// TIA Portal project "Pick & Place XYZ" (V15.1)
// Vorlageprojekt für das Buch mit Zielsystem S7-1200

(* hardware
DEVICE "S7-1200-Station_1"  S7-1200 Station
   slot 0: "Baugruppenträger_0"  Rack  V1.0
   slot 1: "PLC_1"  CPU 1214C DC/DC/DC  6ES7 214-1AG40-0XB0  V4.2
*)

// ===== PLC "PLC_1"  CPU 1214C DC/DC/DC =====

VAR_GLOBAL   // PLC tag table "Standard-Variablentabelle"
   "Transporte_caja" AT %Q0.1 : Bool;
   "Arranque" AT %I0.4 : Bool;
   "Caja_posicion" AT %I0.1 : Bool;
   "X" AT %ID30 : Real;
   "Y" AT %ID34 : Real;
   "Z" AT %ID38 : Real;
   "SPX" AT %QD30 : Real;
   "SPY" AT %QD34 : Real;
   "SPZ" AT %QD38 : Real;
   "Contador_caja" AT %QD42 : DInt;
   "Pallet_posicion" AT %I0.0 : Bool;
   "Sensor_robot" AT %I0.2 : Bool;
   "Sensor_limite-C" AT %I0.3 : Bool;
   "Reset" AT %I0.5 : Bool;
   "Paro" AT %I0.6 : Bool;
   "Paro emergencia" AT %I0.7 : Bool;
   "Automatico" AT %I1.0 : Bool;
   "Factori I/O" AT %I1.1 : Bool;
   "Transpote_pallet" AT %Q0.0 : Bool;
   "Transporte_salida" AT %Q0.2 : Bool;
   "Eje de rotacion" AT %Q0.3 : Bool;
   "Ventosa" AT %Q0.4 : Bool;
   "Baliza verde" AT %Q0.5 : Bool;
   "Baliza amarrila" AT %Q0.6 : Bool;
   "Baliza roja" AT %Q0.7 : Bool;
   "Luz_arranque" AT %Q1.0 : Bool;
   "Luz_reset" AT %Q1.1 : Bool;
   "Luz-paro" AT %Q1.2 : Bool;
   "ET0" AT %M100.0 : Bool;
   "Tag_1" AT %M250.0 : Bool;
   "ET1" AT %M100.1 : Bool;
   "BANDA LIBRE ET" AT %M300.0 : Bool;
   "ET2" AT %M100.2 : Bool;
   "Tag_2" AT %M250.1 : Bool;
   "ET3" AT %M100.3 : Bool;
   "PALLET CPL" AT %M300.1 : Bool;
   "ET4" AT %M100.4 : Bool;
   "ET5" AT %M100.5 : Bool;
   "ET6" AT %M100.6 : Bool;
   "TEMP1" AT %M300.2 : Bool;
   "ET7" AT %M100.7 : Bool;
   "ET8" AT %M101.0 : Bool;
   "ETI" AT %M99.7 : Bool;
   "TIPO CAJA" AT %MW50 : Int;
   "ET9" AT %M101.1 : Bool;
   "ET10" AT %M101.2 : Bool;
   "ET11" AT %M101.3 : Bool;
   "ET12" AT %M101.4 : Bool;
   "ET13" AT %M101.5 : Bool;
   "ET14" AT %M101.6 : Bool;
   "ET15" AT %M101.7 : Bool;
   "ET16" AT %M102.0 : Bool;
   "ET17" AT %M102.1 : Bool;
   "ET20" AT %M102.2 : Bool;
   "ET21" AT %M102.3 : Bool;
   "Tag_3" AT %M250.2 : Bool;
   "TEMP2" AT %M300.3 : Bool;
   "Tag_4" AT %M40.0 : Bool;
   "Marca_Arranque" AT %M60.0 : Bool;
   "Marca_paro" AT %M60.1 : Bool;
   "Marca_emergencia" AT %M60.2 : Bool;
END_VAR

// folder: System blocks/Program resources

DATA_BLOCK "IEC_Timer_0_DB"   // DB1
{ S7_Optimized_Access := 'TRUE' }
AUTHOR : Simatic
FAMILY : IEC
NAME : IEC_TMR
VERSION : 1.0
// stored: InstanceOfName IEC_TIMER
"IEC_TIMER"
BEGIN
END_DATA_BLOCK

DATA_BLOCK "IEC_Counter_0_DB"   // DB2
{ S7_Optimized_Access := 'TRUE' }
AUTHOR : Simatic
FAMILY : IEC
NAME : CNTR
VERSION : 1.0
// stored: InstanceOfName IEC_COUNTER
"IEC_COUNTER"
BEGIN
END_DATA_BLOCK

DATA_BLOCK "IEC_Timer_0_DB_1"   // DB3
{ S7_Optimized_Access := 'TRUE' }
AUTHOR : Simatic
FAMILY : IEC
NAME : IEC_TMR
VERSION : 1.0
// stored: InstanceOfName IEC_TIMER
"IEC_TIMER"
BEGIN
END_DATA_BLOCK

DATA_BLOCK "IEC_Counter_0_DB_1"   // DB4
{ S7_Optimized_Access := 'TRUE' }
AUTHOR : Simatic
FAMILY : IEC
NAME : CNTR
VERSION : 1.0
// stored: InstanceOfName IEC_COUNTER
"IEC_COUNTER"
BEGIN
END_DATA_BLOCK

// folder: (top level)

FUNCTION "MHJ-PLC-Lab-Function-S71200" : Void   // FC9000, SCL
{ S7_Optimized_Access := 'TRUE' }
VERSION : 0.1
   VAR_TEMP
      rdTimeReturn : Int;
      outputTime : DTL;
      SyncVal : Byte;
      forVal : Int;
      forVal_2 : Int;
      Value : Byte;
   END_VAR
   VAR CONSTANT
      CompVal : Byte := 16#34;
      Value_01 : Byte := 16#11;
      Value_01_DW : DWord := 16#A165_D992;
      Value_02_DW : DWord := 16#58BE_4401;
   END_VAR
BEGIN

   #Value:=PEEK(area := 16#82,
        dbNumber := 0,
        byteOffset := 511);
   #Value := #Value + 1;

   POKE(area := 16#82,
        dbNumber := 0,
        byteOffset := 511,
        value := #Value);

   POKE(area:=16#81,
        dbNumber:=0,
        byteOffset:=1016,
        value:=#Value_01_DW);
   POKE(area := 16#81,
        dbNumber := 0,
        byteOffset := 1020,
        value := #Value_02_DW);

   POKE(area := 16#81,
        dbNumber := 0,
        byteOffset := 511,
        value := B#16#00);

   FOR #forVal := 0 TO 120 DO
       FOR #forVal_2:=0 TO 10 DO
           #rdTimeReturn:=RD_SYS_T(#outputTime);
           #rdTimeReturn := WR_SYS_T(#outputTime);
           #rdTimeReturn := RD_SYS_T(#outputTime);
           #rdTimeReturn := WR_SYS_T(#outputTime);
       END_FOR;
       #SyncVal:= PEEK(area := 16#81,
                      dbNumber := 0,
                      byteOffset := 511);
       IF #SyncVal = #CompVal THEN
          GOTO M_1;
       END_IF;
   END_FOR;
   RETURN;

   M_1:
   POKE(area := 16#81,
        dbNumber := 0,
        byteOffset := 511,
        value := B#16#0);
END_FUNCTION

ORGANIZATION_BLOCK "Main"   // OB1, LAD, ProgramCycle
TITLE = "Main Program Sweep (Cycle)"
{ S7_Optimized_Access := 'TRUE' }
VERSION : 0.1
   VAR_INPUT
      Initial_Call : Bool;   // Initial call of this OB
      Remanence : Bool;   // =True, if remanent data are available
   END_VAR
   VAR_TEMP   // added for the SCL form of the ladder/FBD networks
      _w1 : Bool;
      _w2 : Bool;
   END_VAR
BEGIN

REGION Network 1: Konnektierungsbaustein für PLC-Lab
   // Im Netzwerk 1 wird der Konnektierungsbaustein für PLC-Lab aufgerufen.
   // Dieser Aufruf darf nicht entfernt werden!
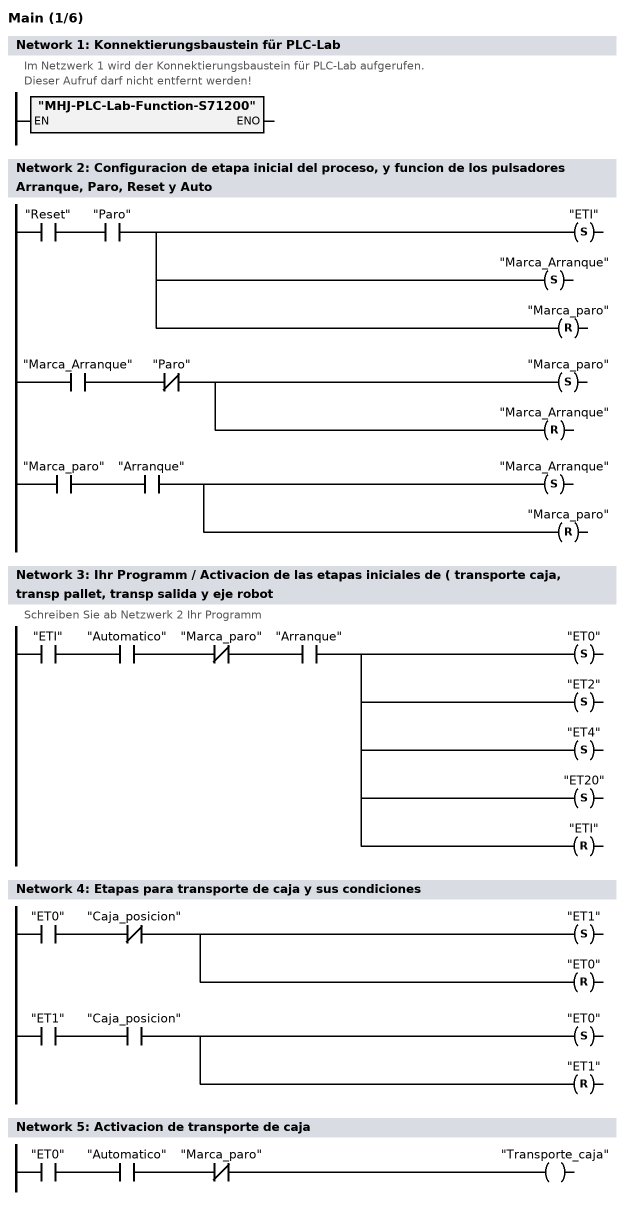
   RUNG wire#powerrail
      "MHJ-PLC-Lab-Function-S71200"()
   END_RUNG
   // the same network as SCL:
   "MHJ-PLC-Lab-Function-S71200"();
END_REGION

REGION Network 2: Configuracion de etapa inicial del proceso, y funcion de los pulsadores Arranque, Paro, Reset y Auto
   RUNG wire#powerrail
      Contact( "Reset" )
      Contact( "Paro" )
      wire#w1
      S_Coil( "ETI" )
   END_RUNG
   RUNG wire#w1
      S_Coil( "Marca_Arranque" )
   END_RUNG
   RUNG wire#w1
      R_Coil( "Marca_paro" )
   END_RUNG
   RUNG wire#powerrail
      Contact( "Marca_Arranque" )
      I_Contact( "Paro" )
      wire#w2
      S_Coil( "Marca_paro" )
   END_RUNG
   RUNG wire#w2
      R_Coil( "Marca_Arranque" )
   END_RUNG
   RUNG wire#powerrail
      Contact( "Marca_paro" )
      Contact( "Arranque" )
      wire#w3
      S_Coil( "Marca_Arranque" )
   END_RUNG
   RUNG wire#w3
      R_Coil( "Marca_paro" )
   END_RUNG
   // the same network as SCL:
   IF "Reset" AND "Paro" THEN
       "ETI" := TRUE;
       "Marca_Arranque" := TRUE;
       "Marca_paro" := FALSE;
   END_IF;
   IF "Marca_Arranque" AND NOT "Paro" THEN
       "Marca_paro" := TRUE;
       "Marca_Arranque" := FALSE;
   END_IF;
   IF "Marca_paro" AND "Arranque" THEN
       "Marca_Arranque" := TRUE;
       "Marca_paro" := FALSE;
   END_IF;
END_REGION

REGION Network 3: Ihr Programm / Activacion de las etapas iniciales de ( transporte caja, transp pallet, transp salida y eje robot
   // Schreiben Sie ab Netzwerk 2 Ihr Programm
   RUNG wire#powerrail
      Contact( "ETI" )
      Contact( "Automatico" )
      I_Contact( "Marca_paro" )
      Contact( "Arranque" )
      wire#w1
      S_Coil( "ET0" )
   END_RUNG
   RUNG wire#w1
      S_Coil( "ET2" )
   END_RUNG
   RUNG wire#w1
      S_Coil( "ET4" )
   END_RUNG
   RUNG wire#w1
      S_Coil( "ET20" )
   END_RUNG
   RUNG wire#w1
      R_Coil( "ETI" )
   END_RUNG
   // the same network as SCL:
   IF "ETI" AND "Automatico" AND NOT "Marca_paro" AND "Arranque" THEN
       "ET0" := TRUE;
       "ET2" := TRUE;
       "ET4" := TRUE;
       "ET20" := TRUE;
       "ETI" := FALSE;
   END_IF;
END_REGION

REGION Network 4: Etapas para transporte de caja y sus condiciones
   RUNG wire#powerrail
      Contact( "ET0" )
      I_Contact( "Caja_posicion" )
      wire#w1
      S_Coil( "ET1" )
   END_RUNG
   RUNG wire#w1
      R_Coil( "ET0" )
   END_RUNG
   RUNG wire#powerrail
      Contact( "ET1" )
      Contact( "Caja_posicion" )
      wire#w2
      S_Coil( "ET0" )
   END_RUNG
   RUNG wire#w2
      R_Coil( "ET1" )
   END_RUNG
   // the same network as SCL:
   IF "ET0" AND NOT "Caja_posicion" THEN
       "ET1" := TRUE;
       "ET0" := FALSE;
   END_IF;
   IF "ET1" AND "Caja_posicion" THEN
       "ET0" := TRUE;
       "ET1" := FALSE;
   END_IF;
END_REGION

REGION Network 5: Activacion de transporte de caja
   RUNG wire#powerrail
      Contact( "ET0" )
      Contact( "Automatico" )
      I_Contact( "Marca_paro" )
      Coil( "Transporte_caja" )
   END_RUNG
   // the same network as SCL:
   "Transporte_caja" := "ET0" AND "Automatico" AND NOT "Marca_paro";
END_REGION

REGION Network 6: Etapas para transporte de pallet y sus condiciones
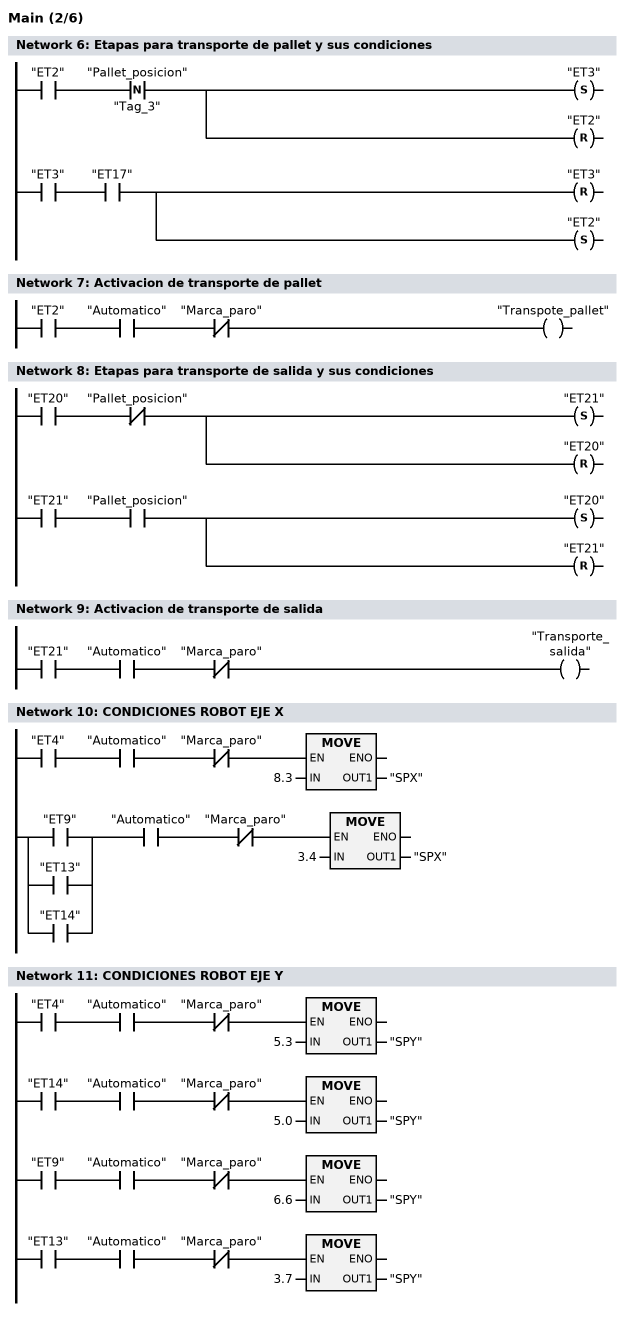
   RUNG wire#powerrail
      Contact( "ET2" )
      N_Contact(operand := "Pallet_posicion", bit := "Tag_3")
      wire#w1
      S_Coil( "ET3" )
   END_RUNG
   RUNG wire#w1
      R_Coil( "ET2" )
   END_RUNG
   RUNG wire#powerrail
      Contact( "ET3" )
      Contact( "ET17" )
      wire#w2
      R_Coil( "ET3" )
   END_RUNG
   RUNG wire#w2
      S_Coil( "ET2" )
   END_RUNG
   // the same network as SCL:
   #_w1 := "ET2" AND NOT "Pallet_posicion" AND "Tag_3";   // falling edge of "Pallet_posicion"
   "Tag_3" := "Pallet_posicion";
   IF #_w1 THEN
       "ET3" := TRUE;
       "ET2" := FALSE;
   END_IF;
   #_w2 := "ET3" AND "ET17";
   IF #_w2 THEN
       "ET3" := FALSE;
       "ET2" := TRUE;
   END_IF;
END_REGION

REGION Network 7: Activacion de transporte de pallet
   RUNG wire#powerrail
      Contact( "ET2" )
      Contact( "Automatico" )
      I_Contact( "Marca_paro" )
      Coil( "Transpote_pallet" )
   END_RUNG
   // the same network as SCL:
   "Transpote_pallet" := "ET2" AND "Automatico" AND NOT "Marca_paro";
END_REGION

REGION Network 8: Etapas para transporte de salida y sus condiciones
   RUNG wire#powerrail
      Contact( "ET20" )
      I_Contact( "Pallet_posicion" )
      wire#w1
      S_Coil( "ET21" )
   END_RUNG
   RUNG wire#w1
      R_Coil( "ET20" )
   END_RUNG
   RUNG wire#powerrail
      Contact( "ET21" )
      Contact( "Pallet_posicion" )
      wire#w2
      S_Coil( "ET20" )
   END_RUNG
   RUNG wire#w2
      R_Coil( "ET21" )
   END_RUNG
   // the same network as SCL:
   IF "ET20" AND NOT "Pallet_posicion" THEN
       "ET21" := TRUE;
       "ET20" := FALSE;
   END_IF;
   IF "ET21" AND "Pallet_posicion" THEN
       "ET20" := TRUE;
       "ET21" := FALSE;
   END_IF;
END_REGION

REGION Network 9: Activacion de transporte de salida
   RUNG wire#powerrail
      Contact( "ET21" )
      Contact( "Automatico" )
      I_Contact( "Marca_paro" )
      Coil( "Transporte_salida" )
   END_RUNG
   // the same network as SCL:
   "Transporte_salida" := "ET21" AND "Automatico" AND NOT "Marca_paro";
END_REGION

REGION Network 10: CONDICIONES ROBOT EJE X
   RUNG wire#powerrail
      Contact( "ET4" )
      Contact( "Automatico" )
      I_Contact( "Marca_paro" )
      Move(in := 8.3, out1 => "SPX")
   END_RUNG
   RUNG wire#powerrail
      Contact( "ET9" )
      wire#w1
      Contact( "Automatico" )
      I_Contact( "Marca_paro" )
      Move(in := 3.4, out1 => "SPX")
   END_RUNG
   RUNG wire#powerrail
      Contact( "ET13" )
   END_RUNG wire#w1
   RUNG wire#powerrail
      Contact( "ET14" )
   END_RUNG wire#w1
   // the same network as SCL:
   IF "ET4" AND "Automatico" AND NOT "Marca_paro" THEN "SPX" := 8.3; END_IF;
   IF ("ET9" OR "ET13" OR "ET14") AND "Automatico" AND NOT "Marca_paro" THEN "SPX" := 3.4; END_IF;
END_REGION

REGION Network 11: CONDICIONES ROBOT EJE Y
   RUNG wire#powerrail
      Contact( "ET4" )
      Contact( "Automatico" )
      I_Contact( "Marca_paro" )
      Move(in := 5.3, out1 => "SPY")
   END_RUNG
   RUNG wire#powerrail
      Contact( "ET14" )
      Contact( "Automatico" )
      I_Contact( "Marca_paro" )
      Move(in := 5.0, out1 => "SPY")
   END_RUNG
   RUNG wire#powerrail
      Contact( "ET9" )
      Contact( "Automatico" )
      I_Contact( "Marca_paro" )
      Move(in := 6.6, out1 => "SPY")
   END_RUNG
   RUNG wire#powerrail
      Contact( "ET13" )
      Contact( "Automatico" )
      I_Contact( "Marca_paro" )
      Move(in := 3.7, out1 => "SPY")
   END_RUNG
   // the same network as SCL:
   IF "ET4" AND "Automatico" AND NOT "Marca_paro" THEN "SPY" := 5.3; END_IF;
   IF "ET14" AND "Automatico" AND NOT "Marca_paro" THEN "SPY" := 5.0; END_IF;
   IF "ET9" AND "Automatico" AND NOT "Marca_paro" THEN "SPY" := 6.6; END_IF;
   IF "ET13" AND "Automatico" AND NOT "Marca_paro" THEN "SPY" := 3.7; END_IF;
END_REGION

REGION Network 12: CONDICIONES EJE Z
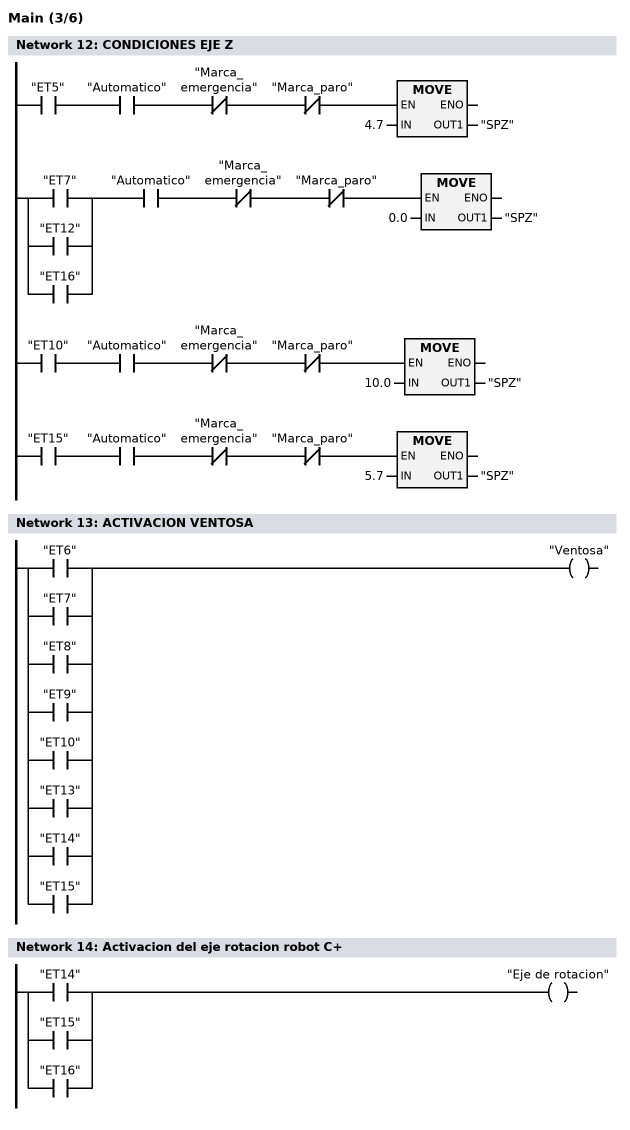
   RUNG wire#powerrail
      Contact( "ET5" )
      Contact( "Automatico" )
      I_Contact( "Marca_emergencia" )
      I_Contact( "Marca_paro" )
      Move(in := 4.7, out1 => "SPZ")
   END_RUNG
   RUNG wire#powerrail
      Contact( "ET7" )
      wire#w1
      Contact( "Automatico" )
      I_Contact( "Marca_emergencia" )
      I_Contact( "Marca_paro" )
      Move(in := 0.0, out1 => "SPZ")
   END_RUNG
   RUNG wire#powerrail
      Contact( "ET12" )
   END_RUNG wire#w1
   RUNG wire#powerrail
      Contact( "ET16" )
   END_RUNG wire#w1
   RUNG wire#powerrail
      Contact( "ET10" )
      Contact( "Automatico" )
      I_Contact( "Marca_emergencia" )
      I_Contact( "Marca_paro" )
      Move(in := 10.0, out1 => "SPZ")
   END_RUNG
   RUNG wire#powerrail
      Contact( "ET15" )
      Contact( "Automatico" )
      I_Contact( "Marca_emergencia" )
      I_Contact( "Marca_paro" )
      Move(in := 5.7, out1 => "SPZ")
   END_RUNG
   // the same network as SCL:
   IF "ET5" AND "Automatico" AND NOT "Marca_emergencia" AND NOT "Marca_paro" THEN "SPZ" := 4.7; END_IF;
   IF ("ET7" OR "ET12" OR "ET16") AND "Automatico" AND NOT "Marca_emergencia" AND NOT "Marca_paro" THEN
       "SPZ" := 0.0;
   END_IF;
   IF "ET10" AND "Automatico" AND NOT "Marca_emergencia" AND NOT "Marca_paro" THEN "SPZ" := 10.0; END_IF;
   IF "ET15" AND "Automatico" AND NOT "Marca_emergencia" AND NOT "Marca_paro" THEN "SPZ" := 5.7; END_IF;
END_REGION

REGION Network 13: ACTIVACION VENTOSA
   RUNG wire#powerrail
      Contact( "ET6" )
      wire#w1
      Coil( "Ventosa" )
   END_RUNG
   RUNG wire#powerrail
      Contact( "ET7" )
   END_RUNG wire#w1
   RUNG wire#powerrail
      Contact( "ET8" )
   END_RUNG wire#w1
   RUNG wire#powerrail
      Contact( "ET9" )
   END_RUNG wire#w1
   RUNG wire#powerrail
      Contact( "ET10" )
   END_RUNG wire#w1
   RUNG wire#powerrail
      Contact( "ET13" )
   END_RUNG wire#w1
   RUNG wire#powerrail
      Contact( "ET14" )
   END_RUNG wire#w1
   RUNG wire#powerrail
      Contact( "ET15" )
   END_RUNG wire#w1
   // the same network as SCL:
   "Ventosa" := "ET6" OR "ET7" OR "ET8" OR "ET9" OR "ET10" OR "ET13" OR "ET14" OR "ET15";
END_REGION

REGION Network 14: Activacion del eje rotacion robot C+
   RUNG wire#powerrail
      Contact( "ET14" )
      wire#w1
      Coil( "Eje de rotacion" )
   END_RUNG
   RUNG wire#powerrail
      Contact( "ET15" )
   END_RUNG wire#w1
   RUNG wire#powerrail
      Contact( "ET16" )
   END_RUNG wire#w1
   // the same network as SCL:
   "Eje de rotacion" := "ET14" OR "ET15" OR "ET16";
END_REGION

REGION Network 15: Activacion de ET5
   // Activacion ET5: Se comprueba de que el robot este en la posicon X=8.3 y Y=5.3 y que las bandas de pallet y caja esten detenidas
   // Activacion ET6: Posicion eje Z=4.7, Sensor de robot activo para succion y activamos un temporizador y se activa ventosa
   // Activacion ET7: Espera temporizador y  ventosa activada
   // Activacion ET8: Se verifica que eje Z=0, ventosa activada
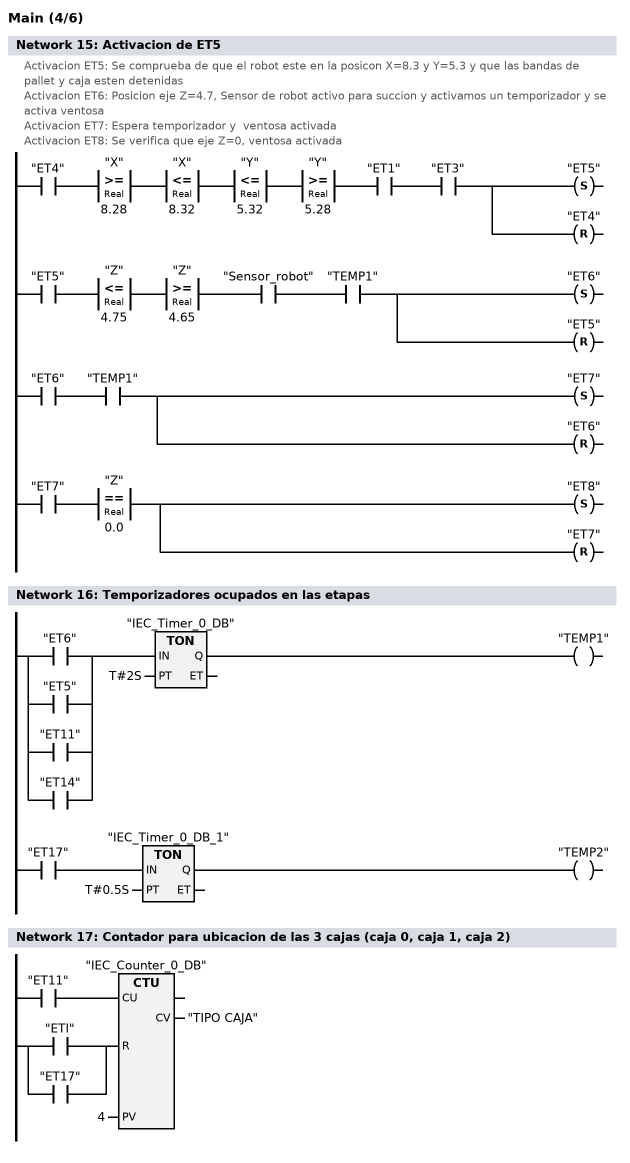
   RUNG wire#powerrail
      Contact( "ET4" )
      { S7_Templates := "SrcType := Real" } GE_Contact(in1 := "X", in2 := 8.28)
      { S7_Templates := "SrcType := Real" } LE_Contact(in1 := "X", in2 := 8.32)
      { S7_Templates := "SrcType := Real" } LE_Contact(in1 := "Y", in2 := 5.32)
      { S7_Templates := "SrcType := Real" } GE_Contact(in1 := "Y", in2 := 5.28)
      Contact( "ET1" )
      Contact( "ET3" )
      wire#w1
      S_Coil( "ET5" )
   END_RUNG
   RUNG wire#w1
      R_Coil( "ET4" )
   END_RUNG
   RUNG wire#powerrail
      Contact( "ET5" )
      { S7_Templates := "SrcType := Real" } LE_Contact(in1 := "Z", in2 := 4.75)
      { S7_Templates := "SrcType := Real" } GE_Contact(in1 := "Z", in2 := 4.65)
      Contact( "Sensor_robot" )
      Contact( "TEMP1" )
      wire#w2
      S_Coil( "ET6" )
   END_RUNG
   RUNG wire#w2
      R_Coil( "ET5" )
   END_RUNG
   RUNG wire#powerrail
      Contact( "ET6" )
      Contact( "TEMP1" )
      wire#w3
      S_Coil( "ET7" )
   END_RUNG
   RUNG wire#w3
      R_Coil( "ET6" )
   END_RUNG
   RUNG wire#powerrail
      Contact( "ET7" )
      { S7_Templates := "SrcType := Real" } EQ_Contact(in1 := "Z", in2 := 0.0)
      wire#w4
      S_Coil( "ET8" )
   END_RUNG
   RUNG wire#w4
      R_Coil( "ET7" )
   END_RUNG
   // the same network as SCL:
   IF "ET4" AND ("X" >= 8.28) AND ("X" <= 8.32) AND ("Y" <= 5.32) AND ("Y" >= 5.28) AND "ET1" AND "ET3" THEN
       "ET5" := TRUE;
       "ET4" := FALSE;
   END_IF;
   IF "ET5" AND ("Z" <= 4.75) AND ("Z" >= 4.65) AND "Sensor_robot" AND "TEMP1" THEN
       "ET6" := TRUE;
       "ET5" := FALSE;
   END_IF;
   IF "ET6" AND "TEMP1" THEN
       "ET7" := TRUE;
       "ET6" := FALSE;
   END_IF;
   IF "ET7" AND ("Z" = 0.0) THEN
       "ET8" := TRUE;
       "ET7" := FALSE;
   END_IF;
END_REGION

REGION Network 16: Temporizadores ocupados en las etapas
   "IEC_Timer_0_DB".TON(IN := "ET6" OR "ET5" OR "ET11" OR "ET14", PT := T#2S);
   "TEMP1" := "IEC_Timer_0_DB".Q;
   "IEC_Timer_0_DB_1".TON(IN := "ET17", PT := T#0.5S);
   "TEMP2" := "IEC_Timer_0_DB_1".Q;
END_REGION

REGION Network 17: Contador para ubicacion de las 3 cajas (caja 0, caja 1, caja 2)
   "IEC_Counter_0_DB".CTU(CU := "ET11", R := "ETI" OR "ET17", PV := 4, CV => "TIPO CAJA");
END_REGION

REGION Network 18: Activacion de las siguientes etapas en dependenica del tipo de caja
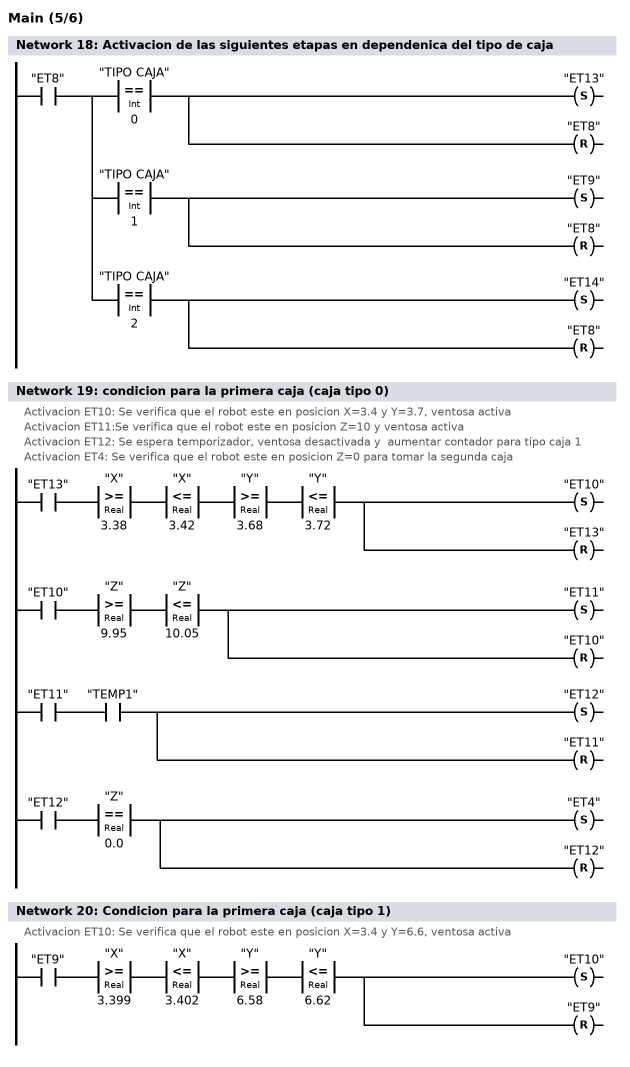
   RUNG wire#powerrail
      Contact( "ET8" )
      wire#w1
      { S7_Templates := "SrcType := Int" } EQ_Contact(in1 := "TIPO CAJA", in2 := 0)
      wire#w2
      S_Coil( "ET13" )
   END_RUNG
   RUNG wire#w2
      R_Coil( "ET8" )
   END_RUNG
   RUNG wire#w1
      { S7_Templates := "SrcType := Int" } EQ_Contact(in1 := "TIPO CAJA", in2 := 1)
      wire#w3
      S_Coil( "ET9" )
   END_RUNG
   RUNG wire#w3
      R_Coil( "ET8" )
   END_RUNG
   RUNG wire#w1
      { S7_Templates := "SrcType := Int" } EQ_Contact(in1 := "TIPO CAJA", in2 := 2)
      wire#w4
      S_Coil( "ET14" )
   END_RUNG
   RUNG wire#w4
      R_Coil( "ET8" )
   END_RUNG
   // the same network as SCL:
   IF "ET8" AND ("TIPO CAJA" = 0) THEN "ET13" := TRUE; END_IF;
   #_w1 := "ET8";
   IF "ET8" AND ("TIPO CAJA" = 0) THEN "ET8" := FALSE; END_IF;
   IF #_w1 AND ("TIPO CAJA" = 1) THEN
       "ET9" := TRUE;
       "ET8" := FALSE;
   END_IF;
   IF #_w1 AND ("TIPO CAJA" = 2) THEN
       "ET14" := TRUE;
       "ET8" := FALSE;
   END_IF;
END_REGION

REGION Network 19: condicion para la primera caja (caja tipo 0)
   // Activacion ET10: Se verifica que el robot este en posicion X=3.4 y Y=3.7, ventosa activa
   // Activacion ET11:Se verifica que el robot este en posicion Z=10 y ventosa activa
   // Activacion ET12: Se espera temporizador, ventosa desactivada y  aumentar contador para tipo caja 1
   // Activacion ET4: Se verifica que el robot este en posicion Z=0 para tomar la segunda caja
   RUNG wire#powerrail
      Contact( "ET13" )
      { S7_Templates := "SrcType := Real" } GE_Contact(in1 := "X", in2 := 3.38)
      { S7_Templates := "SrcType := Real" } LE_Contact(in1 := "X", in2 := 3.42)
      { S7_Templates := "SrcType := Real" } GE_Contact(in1 := "Y", in2 := 3.68)
      { S7_Templates := "SrcType := Real" } LE_Contact(in1 := "Y", in2 := 3.72)
      wire#w1
      S_Coil( "ET10" )
   END_RUNG
   RUNG wire#w1
      R_Coil( "ET13" )
   END_RUNG
   RUNG wire#powerrail
      Contact( "ET10" )
      { S7_Templates := "SrcType := Real" } GE_Contact(in1 := "Z", in2 := 9.95)
      { S7_Templates := "SrcType := Real" } LE_Contact(in1 := "Z", in2 := 10.05)
      wire#w2
      S_Coil( "ET11" )
   END_RUNG
   RUNG wire#w2
      R_Coil( "ET10" )
   END_RUNG
   RUNG wire#powerrail
      Contact( "ET11" )
      Contact( "TEMP1" )
      wire#w3
      S_Coil( "ET12" )
   END_RUNG
   RUNG wire#w3
      R_Coil( "ET11" )
   END_RUNG
   RUNG wire#powerrail
      Contact( "ET12" )
      { S7_Templates := "SrcType := Real" } EQ_Contact(in1 := "Z", in2 := 0.0)
      wire#w4
      S_Coil( "ET4" )
   END_RUNG
   RUNG wire#w4
      R_Coil( "ET12" )
   END_RUNG
   // the same network as SCL:
   IF "ET13" AND ("X" >= 3.38) AND ("X" <= 3.42) AND ("Y" >= 3.68) AND ("Y" <= 3.72) THEN
       "ET10" := TRUE;
       "ET13" := FALSE;
   END_IF;
   IF "ET10" AND ("Z" >= 9.95) AND ("Z" <= 10.05) THEN
       "ET11" := TRUE;
       "ET10" := FALSE;
   END_IF;
   IF "ET11" AND "TEMP1" THEN
       "ET12" := TRUE;
       "ET11" := FALSE;
   END_IF;
   IF "ET12" AND ("Z" = 0.0) THEN
       "ET4" := TRUE;
       "ET12" := FALSE;
   END_IF;
END_REGION

REGION Network 20: Condicion para la primera caja (caja tipo 1)
   // Activacion ET10: Se verifica que el robot este en posicion X=3.4 y Y=6.6, ventosa activa
   RUNG wire#powerrail
      Contact( "ET9" )
      { S7_Templates := "SrcType := Real" } GE_Contact(in1 := "X", in2 := 3.399)
      { S7_Templates := "SrcType := Real" } LE_Contact(in1 := "X", in2 := 3.402)
      { S7_Templates := "SrcType := Real" } GE_Contact(in1 := "Y", in2 := 6.58)
      { S7_Templates := "SrcType := Real" } LE_Contact(in1 := "Y", in2 := 6.62)
      wire#w1
      S_Coil( "ET10" )
   END_RUNG
   RUNG wire#w1
      R_Coil( "ET9" )
   END_RUNG
   // the same network as SCL:
   IF "ET9" AND ("X" >= 3.399) AND ("X" <= 3.402) AND ("Y" >= 6.58) AND ("Y" <= 6.62) THEN
       "ET10" := TRUE;
       "ET9" := FALSE;
   END_IF;
END_REGION

REGION Network 21: Condicion para la primera caja (caja tipo 2)
   // Activacion ET15: Se verifica que el robot este en posicion X=3.4 y Y=5,  sensor de giro activo (limit-c),  temporizador, ademas ventosa activa y  actuador C+ activo
   // Activacion ET16: Se verifica que el robot este en posicion Z=5.7,  actuador C+ activo
   // Activacion ET17: Se verifica que el robot este en posicion Z=0,
   // Activacion ET12: Cumplimiento TEMP2 y  sensor de giro limit-C esta activo, aca se manda a resetear el contador de tipo de caja a tipo caja 0
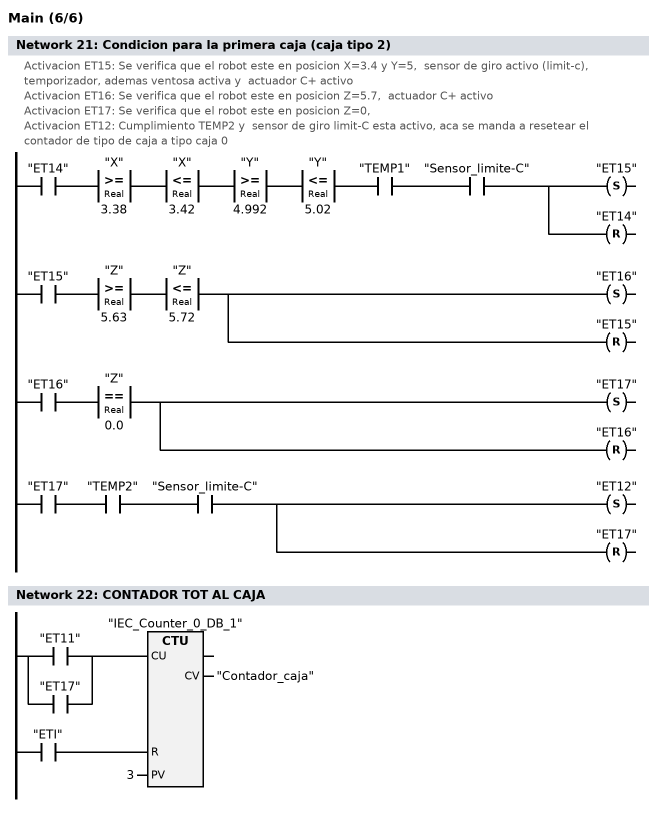
   RUNG wire#powerrail
      Contact( "ET14" )
      { S7_Templates := "SrcType := Real" } GE_Contact(in1 := "X", in2 := 3.38)
      { S7_Templates := "SrcType := Real" } LE_Contact(in1 := "X", in2 := 3.42)
      { S7_Templates := "SrcType := Real" } GE_Contact(in1 := "Y", in2 := 4.992)
      { S7_Templates := "SrcType := Real" } LE_Contact(in1 := "Y", in2 := 5.02)
      Contact( "TEMP1" )
      Contact( "Sensor_limite-C" )
      wire#w1
      S_Coil( "ET15" )
   END_RUNG
   RUNG wire#w1
      R_Coil( "ET14" )
   END_RUNG
   RUNG wire#powerrail
      Contact( "ET15" )
      { S7_Templates := "SrcType := Real" } GE_Contact(in1 := "Z", in2 := 5.63)
      { S7_Templates := "SrcType := Real" } LE_Contact(in1 := "Z", in2 := 5.72)
      wire#w2
      S_Coil( "ET16" )
   END_RUNG
   RUNG wire#w2
      R_Coil( "ET15" )
   END_RUNG
   RUNG wire#powerrail
      Contact( "ET16" )
      { S7_Templates := "SrcType := Real" } EQ_Contact(in1 := "Z", in2 := 0.0)
      wire#w3
      S_Coil( "ET17" )
   END_RUNG
   RUNG wire#w3
      R_Coil( "ET16" )
   END_RUNG
   RUNG wire#powerrail
      Contact( "ET17" )
      Contact( "TEMP2" )
      Contact( "Sensor_limite-C" )
      wire#w4
      S_Coil( "ET12" )
   END_RUNG
   RUNG wire#w4
      R_Coil( "ET17" )
   END_RUNG
   // the same network as SCL:
   IF "ET14" AND ("X" >= 3.38) AND ("X" <= 3.42) AND ("Y" >= 4.992) AND ("Y" <= 5.02) AND "TEMP1" AND "Sensor_limite-C" THEN
       "ET15" := TRUE;
       "ET14" := FALSE;
   END_IF;
   IF "ET15" AND ("Z" >= 5.63) AND ("Z" <= 5.72) THEN
       "ET16" := TRUE;
       "ET15" := FALSE;
   END_IF;
   IF "ET16" AND ("Z" = 0.0) THEN
       "ET17" := TRUE;
       "ET16" := FALSE;
   END_IF;
   IF "ET17" AND "TEMP2" AND "Sensor_limite-C" THEN
       "ET12" := TRUE;
       "ET17" := FALSE;
   END_IF;
END_REGION

REGION Network 22: CONTADOR TOT AL CAJA
   "IEC_Counter_0_DB_1".CTU(CU := "ET11" OR "ET17", R := "ETI", PV := 3, CV => "Contador_caja");
END_REGION
END_ORGANIZATION_BLOCK